FUNCTION_BLOCK Mc2MoveVelocityTask EXTENDS Mc2MotionTask
VAR
	_TargetVelocity : LREAL;
	McMoveVelocity	: ARRAY[0..1] OF Tc2_MC2.MC_MoveVelocity;
	Active			: UDINT;
	_McBufferMode	: Tc2_MC2.MC_BufferMode;
	_MoveOptions	: Tc2_MC2.ST_MoveOptions;
END_VAR

PROPERTY BufferMode : REFERENCE TO MC_BufferMode
GET
BufferMode REF= _McBufferMode;
END_GET
END_PROPERTY

{attribute 'monitoring' := 'call'}
PROPERTY Busy : BOOL
GET
Busy := McMoveVelocity[Active].Busy;
END_GET
END_PROPERTY

METHOD CyclicLogic
VAR
    i : UDINT;
END_VAR
FOR i := 0 TO 1 DO
    McMoveVelocity[i](Axis			:= _Axis.Axis,
                           Velocity		:= _TargetVelocity,
                           Acceleration := _Axis.Acceleration,
                           Deceleration := _Axis.Deceleration,
                           Jerk			:= _Axis.Jerk,
                           BufferMode	:= _McBufferMode,
                           Options		:= _MoveOptions);
    
    McMoveVelocity[i].Execute := FALSE;
END_FOR
END_METHOD

{attribute 'monitoring' := 'call'}
PROPERTY Error : BOOL
GET
Error := McMoveVelocity[Active].Error;
END_GET
END_PROPERTY

{attribute 'monitoring' := 'call'}
PROPERTY ErrorId : UDINT
GET
ErrorID := McMoveVelocity[Active].ErrorID;
END_GET
END_PROPERTY

METHOD Execute : BOOL;
IF _TargetVelocity < 0 THEN
	McMoveVelocity[Active].Direction := MC_Negative_Direction;
ELSE
	McMoveVelocity[Active].Direction := MC_Positive_Direction;
END_IF

_TargetVelocity := ABS(_TargetVelocity);
IF Active = 0 THEN
	Active := 1;
	McMoveVelocity[Active](Axis			:= _Axis.Axis,
						   Execute		:= TRUE,
						   Velocity		:= _TargetVelocity,
						   Acceleration := _Axis.Acceleration,
						   Deceleration := _Axis.Deceleration,
						   Jerk			:= _Axis.Jerk,
						   BufferMode	:= _McBufferMode,
						   Options		:= _MoveOptions);
ELSE
	Active := 0;
	McMoveVelocity[Active](Axis			:= _Axis.Axis,
						   Execute		:= TRUE,
						   Velocity		:= _TargetVelocity,
						   Acceleration := _Axis.Acceleration,
						   Deceleration := _Axis.Deceleration,
						   Jerk			:= _Axis.Jerk,
						   BufferMode	:= _McBufferMode,
						   Options		:= _MoveOptions);
END_IF

Execute := TRUE;
END_METHOD

PROPERTY MoveOptions : REFERENCE TO ST_MoveOptions
GET
MoveOptions REF= _MoveOptions;
END_GET
END_PROPERTY

{attribute 'monitoring' := 'call'}
PROPERTY TargetVelocity : LREAL
SET
_TargetVelocity := TargetVelocity;
END_SET
END_PROPERTY

END_FUNCTION_BLOCK

(* stored: Version 1.1.0.1, ProductVersion 3.1.4026.20
   POU Mc2MoveVelocityTask: Id {80035e3a-ce92-403a-ac1f-ff2608add5d1}, SpecialFunc None
   Property BufferMode: Id {72fd6b5b-0cc6-4cb6-98e8-a852eea2f5cd}
   Get Get: Id {487b478e-be24-4e0f-8270-ff012b3ee207}
   Property Busy: Id {6a44be82-2189-44dd-8de7-d4602b0d72d6}
   Get Get: Id {9160f6ac-d9da-45a5-a137-d461f446b744}
   Method CyclicLogic: Id {d50165cf-a947-4fb6-bb92-bba9143099c2}
   Property Error: Id {7413c3d1-d094-459e-a74f-5e05ede91922}
   Get Get: Id {81b7a07a-b770-4454-bea1-25574171c82d}
   Property ErrorId: Id {1002ce08-94ad-4987-aa50-d81de84f78f4}
   Get Get: Id {1119a231-53c2-451a-bee2-c43af74bde02}
   Method Execute: Id {fa35fd38-9981-40a9-b84b-6eb8b7b264e1}
   Property MoveOptions: Id {f39363c6-5cb9-4a87-89b3-95cb5a4df2e1}
   Get Get: Id {536f92d0-809e-4457-a511-f209223944ba}
   Property TargetVelocity: Id {3e5a7470-c459-462c-bf5f-0a4a0a464803}
   Set Set: Id {16e5e7dd-2a64-44fc-91b2-8e34f4175d40} *)
